TYPE u_SM6020_temp :
UNION
	temp	:ARRAY[0..1] OF BYTE;
	itemp			:INT;
END_UNION
END_TYPE

(* stored: Version 1.1.0.1, ProductVersion 3.1.4024.12
   DUT u_SM6020_temp: Id {ea5a7fa2-edaa-4f26-9d8f-f24e0403f695} *)
